FUNCTION_BLOCK KeyValueCollectionDisposedEventHandler EXTENDS KeyValueCollectionEventHandler

METHOD PUBLIC HandleEvent
VAR_INPUT
	Event : I_Event;
END_VAR
VAR
	disposedEvent : I_KeyValueCollectionDisposedEvent;
END_VAR
IF __QUERYINTERFACE(Event, disposedEvent) THEN
	_eventReceived := TRUE;
	fromExpected := disposedEvent.Target = expectedOriginator;
END_IF
END_METHOD

END_FUNCTION_BLOCK

(* stored: Version 1.1.0.1, ProductVersion 3.1.4024.12
   POU KeyValueCollectionDisposedEventHandler: Id {4f327b1d-2b0e-4e18-bf6d-0472e395c6b1}, SpecialFunc None
   Method HandleEvent: Id {6a30c584-7c49-4ded-96fc-da444446ed5c} *)
